				0: // Start-up/Init
					IF fbPlanarXtsMover.P_MoverSort.TrackID = GVL_General.PlanarTrackOuterFinish THEN
						fbPlanarXtsMover.P_MC_PlanarMover.MoveOnTrack(commandFeedback := fbPlanarXtsMover.P_MoverFeedback,
																			targetTrack := GVL_Mc3.MC_Tracks[E_TrackNum.Big],
																			targetPositionOnTrack := GVL_Mc3.MC_Tracks[E_TrackNum.Big].GetLength()-stTrackGlobalConfig.TargetPosnBeforeTrackEnd,
																			constraint := fbPlanarXtsMover.P_Dynamics,
																			options := fbPlanarXtsMover.P_MoverOptions.BaseMoveOptions);
						 nMoveState 	:= 20;
					ELSIF (fbPlanarXtsMover.P_MoverSort.TrackID = GVL_General.PlanarTrackOuterStart) AND 
								fbPlanarXtsMover.P_XtsPositionInfo.fPartPosition < TrackSectors.P_SectorsConfig[GC.DIVERTQ_SECTOR_OPART].PartSectorStartPosn THEN
						fbPlanarXtsMover.P_MC_PlanarMover.MoveOnTrack(commandFeedback := fbPlanarXtsMover.P_MoverFeedback,
																			targetTrack := GVL_Mc3.MC_Tracks[E_TrackNum.Main],
																			targetPositionOnTrack := GVL_Mc3.MC_Tracks[E_TrackNum.Main].GetLength()-stTrackGlobalConfig.TargetPosnBeforeTrackEnd,
																			constraint := fbPlanarXtsMover.P_Dynamics,
																			options := fbPlanarXtsMover.P_MoverOptions.BaseMoveOptions);
						 nMoveState 	:= 10;
					END_IF
					
				5: // In Recirc - from Big to Main Track - departing Gap Transition Zone - this Move command could be cyclic
					IF stPlcSystem.TempSysTime = 0 XOR stPlcSystem.TempSysTime = stPlcSystem.SysTime THEN
						stPlcSystem.TempSysTime := stPlcSystem.SysTime + (stPlcSystem.CfgIntervalExec * stPlcSystem.nCycleTime); //next valid clock to issue move command again
						fbPlanarXtsMover.P_eMerge		:= E_MergeType.NoMerge;
						fbPlanarXtsMover.P_MasterSyncId	:= 0;
						fbPlanarXtsMover.P_MasterSyncPosition	:= 0;
						fbPlanarXtsMover.P_MC_PlanarMover.MoveOnTrack(commandFeedback := fbPlanarXtsMover.P_MoverFeedback,
																		targetTrack := GVL_Mc3.MC_Tracks[E_TrackNum.Main],
																		targetPositionOnTrack := GVL_Mc3.MC_Tracks[E_TrackNum.Main].GetLength()-stTrackGlobalConfig.TargetPosnBeforeTrackEnd,
																		constraint := fbPlanarXtsMover.P_Dynamics, 
																		options := fbPlanarXtsMover.P_MoverOptions.BaseMoveOptions);
					END_IF
																		
					//Continuously call the above move command while GapInTransition TRUE (otherwise it's a one-shot command)
					IF NOT fbPlanarXtsMover.P_MoverOptions.GapInTransition THEN
						stPlcSystem.TempSysTime		:= 0;
						nMoveState 	:= 10;
					END_IF

				10: //Trig state for decision to divert
					IF TrackSectors.afbSector[GC.DIVERTQ_SECTOR_OPART].stSectorStatus.MoverEnteredSector.Q THEN
						GVL_General.stSwitchStatus.ShuttleCountAtDivertTrig		:= GVL_General.stSwitchStatus.ShuttleCountAtDivertTrig +1; //always MODing this; don't need to decrement
						TempItvlMoverIndex	:= ((GVL_General.stSwitchStatus.ShuttleCountAtDivertTrig MOD GVL_General.stSwitchConfig.SwitchModeInternal.IntervalToDivert) +1); // capture the index
					//	AllTrackSectors.M_UpdateSectorCounts(SectorNr := GC.SHORTCUT_CALC_SECTOR_IPART);
						MoverIndexDivertTrig			:= fbPlanarXtsMover.P_MoverId; // regardless of the command to divert, log the MoverID
						DivertQueue.M_UpdateAtTrig();
						nMoveState 	:= 12;
					END_IF
					
				12: // Command to move needs to be given early
					IF TrackSectors.afbSector[GC.DIVERT_DECISION_OPART].stSectorStatus.MoverEnteredSector.Q THEN
						DivertQueue.RemoveObjFromBuffer();
						nMoveState 	:= 13;
					END_IF
				
				13:				
				IF (DivertQueue.P_LastObjectRemoved.MoverID <> 0) THEN // Valid MoverID must be obtained by Remove op in previous step
					IF SwitchMagnet.P_PermIntlkOK AND NOT MagnetControlledByOtherMover AND fbPlanarXtsMover.P_CmdDivert AND 
						(fbPlanarXtsMover.P_XtsPositionInfo.fPartPosition < GVL_Mc3.TrackSectors.P_SectorConfig[GC.MAG_ON_SECTOR_OPART].PartSectorStartPosn)
						AND (stDivertingMover.SysTime <> DivertQueue.P_LastObjectRemoved.SysTime) THEN
							// Divert Move command
							stDivertingMover	:= DivertQueue.P_LastObjectRemoved;
							fbPlanarXtsMover[stDivertingMover.MoverID].P_MC_PlanarMover.MoveOnTrack(commandFeedback := fbPlanarXtsMover[stDivertingMover.MoverID].P_MoverFeedback,
																				targetTrack := GVL_Mc3.MC_Tracks[E_TrackNum.Small],
																				targetPositionOnTrack := (GVL_Mc3.MC_Tracks[E_TrackNum.Small].GetLength() - GC.SHUTTLE_LENGTH) / 2, // midpoint of shortcut
																				constraint := fbPlanarXtsMover[stDivertingMover.MoverID].P_Dynamics,
																				options := fbPlanarXtsMover[stDivertingMover.MoverID].P_MoverOptions.BaseMoveOptions);									
							nMoveState 	:= 30; //Diverting Mover
					ELSIF NOT fbPlanarXtsMover.P_CmdDivert THEN
							nMoveState 	:= 15;
					END_IF
				END_IF
	
				15: // In Recirc - from Main to Big Track
					fbPlanarXtsMover.P_MC_PlanarMover.MoveOnTrack(commandFeedback := fbPlanarXtsMover.P_MoverFeedback,
																		targetTrack := GVL_Mc3.MC_Tracks[E_TrackNum.Big],
																		targetPositionOnTrack := GVL_Mc3.MC_Tracks[E_TrackNum.Big].GetLength()-stTrackGlobalConfig.TargetPosnBeforeTrackEnd,
																		constraint := fbPlanarXtsMover.P_Dynamics,
																		options := fbPlanarXtsMover.P_MoverOptions.BaseMoveOptions);
					 nMoveState 	:= 20;				
					
				20:
					IF TrackSectors.afbSector[GC.OUTER_BIGTRACK_END].stSectorStatus.MoverEnteredSector.Q THEN
						nMoveState     := 5;
					END_IF				

				30: // Match the move command with the shuttle that is commanded to divert
					SwitchMagnet.M_EvaluateInlineCommands();
					
					IF ftMagnetControlledByOtherMover.Q THEN
						nMoveState 	:= 40;
					END_IF
			
				40: // Route through shortcut
					IF TrackSectors.afbSector[GC.LOAD_STOP_SECTOR_IPART].stSectorStatus.MoverEnteredSector.Q THEN
						IF stTrackShortcutConfig.StopAtPowerMat THEN
							nMoveState := 90;
						ELSE
							nMoveState := 50;
						END_IF					
					END_IF
					
				50: //Pre-Merge state
				IF NOT AllTrackSectors.P_AMoverIsOnSector[GC.OUTER_BIGTRACK_LSMALL] 
						(*AND stSwitchConfig.SwitchModeInternal.MaxAllowedDivertCount = GVL_General.nNumMovers*) THEN
					fbPlanarXtsMover.P_eMerge := E_MergeType.FlyingMergeMoveOnTrack;

					fbPlanarXtsMover.P_MC_PlanarMover.MoveOnTrack(commandFeedback := fbPlanarXtsMover.P_MoverFeedback,
																		targetTrack := GVL_Mc3.MC_Tracks[E_TrackNum.Small],
																		targetPositionOnTrack := GVL_Mc3.MC_Tracks[E_TrackNum.Small].GetLength()-stTrackGlobalConfig.TargetPosnBeforeTrackEnd,
																		constraint := fbPlanarXtsMover.P_Dynamics,
																		options := fbPlanarXtsMover.P_MoverOptions.BaseMoveOptions);

					nMoveState := 75;
					//Sync to Master ExpMover
				ELSIF TrackSectors.afbSector[GC.SHORTCUT_MERGE_COMMAND_FLYING].stSectorStatus.MoverEnteredSector.Q THEN
					//Nonzero means there is valid Master Mover data
					IF MergeQueue.P_LastObjectRemoved.MoverID <> 0 THEN
					fbPlanarXtsMover.P_eMerge				:= E_MergeType.FlyingMergeMoveSyncd;
						fbPlanarXtsMover.P_MasterSyncId := MergeQueue.P_LastObjectRemoved.MoverID;
//						IF MergeQueue.P_LastObjectRemoved.ExpMoverType = E_ExpMover.Head THEN
//							fbPlanarXtsMover.P_MasterSyncPosition	:= HeadExpMover[fbPlanarXtsMover.P_MasterSyncId].stExpMoverStatus.TrackSectorCenterHead;
//						ELSIF MergeQueue.P_LastObjectRemoved.ExpMoverType = E_ExpMover.Tail THEN
//							fbPlanarXtsMover.P_MasterSyncPosition	:= TailExpMover[fbPlanarXtsMover.P_MasterSyncId].stExpMoverStatus.TrackSectorCenterTail;
//						END_IF
							// use raw mover reference; likely need some position compensation, i.e, stTrackGlobalConfig.ExpMoverLength;
							fbPlanarXtsMover.P_MasterSyncPosition	:= fbPlanarXtsMover[fbPlanarXtsMover.P_MasterSyncId].P_XtsPositionInfo.fTrackPosition;							
						MergeQueue.ClearLastRemoved(); // master sync data consumed by slave
						nMoveState := 72;					
					END_IF
					
				ELSIF TrackSectors.afbSector[GC.SHORTCUT_MERGE_COMMAND_WAIT].stSectorStatus.MoverEnteredSector.Q OR 
					stTrackShortcutConfig.StopAtPowerMat THEN
					fbPlanarXtsMover.P_eMerge := E_MergeType.MergeFromStaticSyncd;
					
					fbPlanarXtsMover.P_MC_PlanarMover.MoveOnTrack(commandFeedback := fbPlanarXtsMover.P_MoverFeedback,
																		targetTrack := GVL_Mc3.MC_Tracks[E_TrackNum.Small],
																		targetPositionOnTrack := GVL_Mc3.MC_Tracks[E_TrackNum.Small].GetLength()-stTrackGlobalConfig.MergeWaitFinishDistance-stTrackGlobalConfig.MergeWaitAccelDistance,
																		constraint := fbPlanarXtsMover.P_Dynamics,
																		options := fbPlanarXtsMover.P_MoverOptions.BaseMoveOptions);

					nMoveState := 73;
				END_IF

				60: // Merge - Gear In
 //merge with gap zero
					//issue commmand to sync 
//					masterSyncPos := GVL_Mc.MC_Tracks[E_TrackNum.Big].GetLength()-100;
//					masterPosAtSync := Mover[moverInFront].MoverPos; 
//					followSyncPos := GVL_Mc.MC_Tracks[E_TrackNum.Small].GetLength()-1000;
//					followerPosAtSync :=Mover[1].MoverPos; 
//					fbMover[nForCounter].SyncToOtherMover( 
//						masterSyncPos := masterSyncPos,
//						masterTrack := GVL_Mc.MC_Tracks[E_TrackNum.Big],
//						followerSyncPos := followSyncPos,
//						followerTrack := GVL_Mc.MC_Tracks[e_TrackNum.Small],
//						PlanarMoverToFollow := fbMover[moverInFront].P_PlanarMover,
//						velo:= velo);
//						nMoveState := 80; 
//					aggressiveDynamics.SetValuesVADJ(4000,4000,8000,400000); 
//					fbMover[nForCounter].P_Dynamics := aggressiveDynamics;
					//fbMover[nForCounter].MoveOnTrack(GVL_Mc.MC_Tracks[E_TrackNum.Main],  GVL_Mc.MC_Tracks[E_TrackNum.Main].GetLength()-500,900,velo);				
				
//					IF fbPlanarXtsMover.P_eMerge <> E_MergeType.NoMerge THEN
						fbPlanarXtsMover.P_Dynamics.SetValuesVADJ(V := stMoverConfig.NormalVelo, A := stMoverConfig.MaxAccel, D := stMoverConfig.MaxDecel, J := stMoverConfig.MergeJerk);
						
						fbPlanarXtsMover.P_MC_PlanarMover.GearInPosOnTrackWithMasterMover(
								commandFeedback:= fbPlanarXtsMover.P_PlanarFeedbackGearMM, 
								masterMover:= fbPlanarXtsMover[fbPlanarXtsMover.P_MasterSyncId].P_MC_PlanarMover,
								trackTrail:= fbPlanarXtsMover.P_SyncTrail,
								masterSyncPosition:= fbPlanarXtsMover.P_MasterSyncPosition,
								masterSyncPositionTrack:= GVL_Mc3.MC_Tracks[E_TrackNum.Big], 
								slaveSyncPosition:= fbPlanarXtsMover.P_XtsPositionInfo.fTrackPosition,
								slaveSyncPositionTrack:= GVL_Mc3.MC_Tracks[E_TrackNum.Small], 
								constraint:= fbPlanarXtsMover.P_Dynamics, 
								options:= fbPlanarXtsMover.P_MoverOptions.GearInMasterMoverOptions);
								nMoveState := 74;
//					END_IF
						//fbPlanarXtsMover.P_InSync THEN				

				61:
				IF fbPlanarXtsMover.P_MoverFeedback.Done AND ManMergeCmd THEN
					ManMergeCmd	:= FALSE;
					nMoveState := 75; // 62
				END_IF
					
				62:// Permissive to Merge
//					IF NOT AllTrackSectors.P_AMoverIsOnSector[GC.OUTER_MERGE_COLLISION] THEN
//						nMoveState := 63;
//					END_IF

				63://Merge from Inner to Outer
//						fbPlanarXtsMover.P_MC_PlanarMover.MoveOnTrack(commandFeedback := fbPlanarXtsMover.P_MoverFeedback,
//																			targetTrack := GVL_Mc3.MC_Tracks[E_TrackNum.Small],
//																			targetPositionOnTrack := GVL_Mc3.MC_Tracks[E_TrackNum.Small].GetLength()-stTrackGlobalConfig.TargetPosnBeforeTrackEnd,
//																			constraint := fbPlanarXtsMover.P_Dynamics,
//																			options := fbPlanarXtsMover.P_MoverOptions.BaseMoveOptions);
//						nMoveState := 75;
				
				75: //Reset Command On Exit
						IF TrackSectors.afbSector[GC.INNER_MERGE_TO_FINISH].stSectorStatus.MoverEnteredSector.Q THEN
							stSwitchStatus.ShuttleQueueCount := stSwitchStatus.ShuttleQueueCount -1;
							nMoveState := 5;
						END_IF
				
				90: // Stopped at Powermat Station
					IF fbPlanarXtsMover.P_MoverFeedback.Done THEN
						StartTimer[nForCounter] := TRUE;
						nMoveState := 100;
					END_IF
					
				100:
					IF StopTimer[nForCounter].Q THEN
						StartTimer[nForCounter] := FALSE;
						nMoveState := 50;
					END_IF
				END_CASE
				*)

METHOD M_EvaluateTrackTransition
VAR_INPUT
	DepartingTrackRef : OTCID;
	ArrivingTrackRef : OTCID;
	DepartPermissiveSectorRef	: UDINT;
END_VAR
END_METHOD

END_FUNCTION_BLOCK

// ---- POUs/FBs/FB_RobMover.TcPOU
{attribute 'no_assign'}
FUNCTION_BLOCK FB_RobMover IMPLEMENTS I_Mover
VAR_INPUT
END_VAR
VAR_OUTPUT
END_VAR
VAR
	fbPlanarMover : MC_PlanarMover;
	fbPlanarFeedback: MC_PlanarFeedback;
	CmdFeedback :  XtsCommandFeedback;
	bIsInitialized: BOOL;
	ipXtsMover:   I_XtsXlMover1;
	ipXtsProcessingUnit:  I_XtsProcessingUnit1;
	trackTrail: MC_PlanarTrackTrail;
	nextMcTrackOid: OTCID;
	stMoveOnTrackOptions: ST_MoveOnTrackOptions;
	_stDynamics: DynamicConstraint_PathXY;
	_TargetTrack : UDINT;
	_ReWork : BOOL;
	partConfig1: UINT;
	SyncMoverFeedback: Tc3_Mc3PlanarMotion.MC_PlanarFeedbackGearInPosOnTrackWithMasterMover;
	_InSync :BOOL; 
	options: Tc3_Mc3PlanarMotion.ST_GearInPosOnTrackWithMasterMoverOptions;
	syncTrail : MC_PlanarTrackTrail; 
END_VAR

METHOD CycleUpdate : BOOL
VAR_INPUT
END_VAR
IF NOT bIsInitialized THEN
	RETURN;
END_IF

fbPlanarMover.GetTrackTrailInformation(trackTrail);


fbPlanarMover.Update();


fbPlanarFeedback.Update();
SyncMoverFeedback.Update(); 
_InSync := SyncMoverFeedback.inSync; 

UpdateXtsTrack();
END_METHOD

METHOD Init : BOOL
VAR_INPUT

	XtsMover:   I_XtsXlMover1;
	XtsProcessingUnit :  I_XtsProcessingUnit1;
END_VAR



ipXtsMover:= XtsMover;
ipXtsProcessingUnit :=  XtsProcessingUnit;

stMoveOnTrackOptions.direction := MC_Direction.mcDirectionPositive;
stMoveOnTrackOptions.gapMode := MC_GAP_MODE_ON_TRACK.Fast1D;
stMoveOnTrackOptions.gap:= 800;

syncTrail.AddTrack(track:= GVL_Mc.MC_Tracks[E_TrackNum.Small]); 
syncTrail.AddTrack(track:= GVL_Mc.MC_Tracks[E_TrackNum.Main]); 


//_stDynamics.SetValuesVADJ(500, 4000, 4000, 10000);

bIsInitialized := TRUE;
END_METHOD

METHOD JoinNearestTrack : BOOL


VAR_INST
	nForCounter: UINT;
	mcTrackOid: OTCID;
	partOid: OTCID;
	cmdFeedback					: 	XtsCommandFeedback;
	objectInfo: PlanarObjectInfo;
END_VAR
partOid := ipXtsMover.GetPositionInfo_partObjectId(cmdFeedback);

IF partOid = 0 THEN
	RETURN;
END_IF

IF cmdFeedback.IsDone THEN
	mcTrackOid := ipXtsProcessingUnit.XlPartWithOid(partOid, cmdFeedback).GetMcTrackOid(cmdFeedback);
	
	FOR nForCounter := 1 TO GVL_MC.nTrackCount DO
		objectInfo := GVL_MC.Mc_Tracks[nForCounter].GetPlanarObjectInfo();
		IF objectInfo.Id = mcTrackOid THEN
			fbPlanarMover.JoinTrack(fbPlanarFeedback, GVL_MC.Mc_Tracks[nForCounter], _stDynamics, 0); 
			RETURN;
		END_IF
	END_FOR
END_IF
END_METHOD

METHOD LeaveSystemAt : BOOL
VAR_INPUT
	ConnectionOut: REFERENCE TO MC_PlanarTrackConnectionOut;
END_VAR
fbPlanarMover.LeaveSystemAt(fbPlanarFeedback, ConnectionOut,  _stDynamics,0);
END_METHOD

METHOD MoveOnTrack : BOOL
VAR_INPUT
	
	track: REFERENCE TO MC_PlanarTrack;	
	targetPos: LREAL;
	gap : LREAL; 
	velo : LREAL; 
END_VAR
stMoveonTrackOptions.gap := gap; 
THIS^.P_Dynamics.V := velo; 
fbPlanarMover.MoveOnTrack(fbPlanarFeedback, track, targetPos, _stDynamics, stMoveOnTrackOptions);
END_METHOD

PROPERTY MoverOTCID : OTCID
GET
MoverOTCID := fbPlanarMover.MCTOPLC.STD.MoverOID;
END_GET
SET
END_SET
END_PROPERTY

PROPERTY MoverStopped : BOOL
GET
MoverStopped := (fbPlanarMover.MCTOPLC.SETONTRACK.SetVelo < 20);
END_GET
SET
END_SET
END_PROPERTY

PROPERTY P_Dynamics : REFERENCE TO DynamicConstraint_PathXY;
GET

P_Dynamics REF= _stDynamics;
END_GET
SET // PUBLIC
_stDynamics := P_Dynamics;
END_SET
END_PROPERTY

PROPERTY P_InSync : Bool
GET
P_InSync := _InSync;
END_GET
END_PROPERTY

PROPERTY P_PlanarFeedback : REFERENCE TO MC_PlanarFeedback
GET
P_PlanarFeedback REF= fbPlanarFeedback;
END_GET
END_PROPERTY

PROPERTY P_PlanarMover :   REFERENCE TO  MC_PlanarMover
GET
P_PlanarMover REF= fbPlanarMover;
END_GET
END_PROPERTY

PROPERTY P_TargetTrack : UDINT
GET
P_TargetTrack := _TargetTrack ;
END_GET
SET
_TargetTrack := P_TargetTrack;
END_SET
END_PROPERTY

PROPERTY Rework : BOOL
GET
Rework := _Rework;
END_GET
SET
_Rework := Rework;
END_SET
END_PROPERTY

METHOD SyncToOtherMover : BOOL
VAR_INPUT
	masterSyncPos : LREAL; // Position on the master track
	followerSyncPos : LREAL; // position on the follower track
	PlanarMoverToFollow: REFERENCE TO Tc3_Mc3PlanarMotion.MC_PlanarMover;
	masterTrack : REFERENCE TO Tc3_Mc3PlanarMotion.MC_PlanarTrack; 
	followerTrack : REFERENCE TO Tc3_Mc3PlanarMotion.MC_PlanarTrack; 
	velo : LREAL; 
END_VAR

VAR
	trail: Tc3_Mc3PlanarMotion.MC_PlanarTrackTrail;

END_VAR
Options.allowedSlaveSyncDirections := MC_SYNC_DIRECTIONS.Positive; 
options.directionMasterSyncPosition := MC_DIRECTION.mcDirectionNonModulo; 
options.directionSlaveSyncPosition := MC_DIRECTION.mcDirectionNonModulo;  
options.followMover := FALSE; 
options.gap := 0; // elimnate gap funciton 
options.inSyncToleranceDistance :=0; 
options.moduloToleranceMasterSyncPosition := 0; 
options.moduloToleranceSlaveSyncPosition := 0;  
_stDynamics.V := velo; 

fbPlanarMover.GearInPosOnTrackWithMasterMover(
	commandFeedback:=  SyncMoverFeedback , 
	masterMover:= PlanarMoverToFollow , 
	trackTrail:= syncTrail, // may need to give a trail maybe not
	masterSyncPosition:= masterSyncPos, 
	masterSyncPositionTrack:= MasterTrack , 
	slaveSyncPosition:= followerSyncPos, 
	slaveSyncPositionTrack:= followerTrack, 
	constraint:=_stDynamics , 
	options:=options );
END_METHOD

METHOD PUBLIC UpdateXtsTrack
VAR_INPUT
END_VAR
VAR_STAT
	nTrackCount: UINT;
	oid1: OTCID;
	oid2: OTCID;
	
	nForCounter: UINT;
	nPartConfigCount: UINT;
	
	partConfig1: OTCID;
	partConfig2: OTCID;
	
	mcTrackOid1: OTCID;
	mcTrackOid2: OTCID;
	trackOid: OTCID;
	
	nTrackTrailCount: UDINT;
	actTrackOid: OTCID;
	nIndexInTrail: UDINT;
END_VAR
nTrackTrailCount := trackTrail.TrackCount;
actTrackOid := fbPlanarMover.MCTOPLC.SETONTRACK.TrackOID;

IF nTrackTrailCount <= 1 THEN
	RETURN;
END_IF

FOR nForCounter := 1 TO UDINT_TO_UINT(nTrackTrailCount) DO
	oid1 := trackTrail.GetTrackOidAt(nForCounter);
	IF oid1 = actTrackOid THEN
		IF nForCounter < nTrackTrailCount THEN
			oid2 := trackTrail.GetTrackOidAt(nForCounter + 1);
			EXIT;
		ELSE
			RETURN; //last one ine track trail
		END_IF
	END_IF
END_FOR

IF oid2 = nextMcTrackOid AND   ipXtsMover.GetPositionInfo_partPosition(CmdFeedback) < 600THEN //no change
	RETURN;
END_IF

nTrackCount := ipXtsProcessingUnit.TrackCount();

FOR nForCounter := 1 TO nTrackCount DO
	nPartConfigCount := ipXtsProcessingUnit.Track(nForCounter, CmdFeedback).PartConfigCount(); 
	
	IF nPartConfigCount >= 2  THEN
		partConfig1 := ipXtsProcessingUnit.Track(nForCounter, CmdFeedback).GetPartConfigOidAt(1, 0);
		partConfig2 := ipXtsProcessingUnit.Track(nForCounter, CmdFeedback).GetPartConfigOidAt(2, 0);
//
		
		IF partConfig1 = 0 OR partConfig2 = 0 THEN
			CONTINUE;
		END_IF
		
		mcTrackOid1 := ipXtsProcessingUnit.XlPartWithOid(partConfig1, CmdFeedback).GetMcTrackOid(0);
		mcTrackOid2 := ipXtsProcessingUnit.XlPartWithOid(partConfig2, CmdFeedback).GetMcTrackOid(0);
		IF mcTrackOid1 = oid1 AND mcTrackOid2 = oid2   THEN
			trackOid := ipXtsProcessingUnit.Track(nForCounter, CmdFeedback).GetObjectId();
			ipXtsMover.SetActiveTrackObjectId(trackOid, CmdFeedback);
			
			IF CmdFeedback.IsDone THEN
				nextMcTrackOid := oid2;
			END_IF
			
			RETURN;
		END_IF
	END_IF
END_FOR
END_METHOD

PROPERTY XlProcessingUnit : I_XtsProcessingUnit1
GET
XlProcessingUnit := ipXtsProcessingUnit;
END_GET
END_PROPERTY

PROPERTY XtsComFeed : REFERENCE TO  XtsCommandFeedback
GET
XtsComFeed REF= CmdFeedback;
END_GET
END_PROPERTY

PROPERTY XtsXlMover : I_XtsXlMover1
GET
XtsXlMover := ipXtsMover;
END_GET
END_PROPERTY

END_FUNCTION_BLOCK

// ---- POUs/FBs/ReadTcCom.TcPOU
FUNCTION_BLOCK ReadTcCom
VAR_INPUT
	
END_VAR
VAR_OUTPUT
	bBusy 				: BOOL;
	bDone 				: BOOL;
	bError 				: BOOL;
	bGetComObject	: BOOL;
END_VAR
VAR
	
	_nObjectId				: OTCID;
	_ipComObject 			: ITComObject;
	_nSoftDriveOid			: OTCID;
	PID_Value	: PTCID := 	16#05030149;
END_VAR

METHOD GetComObject : BOOL
VAR_INPUT
	nObjectId	: OTCID;
END_VAR
IF FW_ObjMgr_GetObjectInstance(	oid		:= nObjectId, 
								iid		:= TC_GLOBAL_IID_LIST.IID_ITComObject, 
								pipUnk	:= ADR(_ipComObject)) = 0
THEN
	GetComObject := TRUE;
END_IF
END_METHOD

METHOD GetValue : ARRAY[1..nNumMovers] OF OTCID
VAR_INPUT
	PID_Value 		: otcid;
END_VAR
VAR
	Value			: ARRAY[1..nNumMovers] OF OTCID;
	nData 			: UDINT := SIZEOF(Value);
	pData 			: PVOID := ADR(Value);
	stEventEntry	: TcEventEntry;
	pstEventEntry	: REFERENCE TO TcEventEntry REF= stEventEntry;
	
END_VAR
VAR_INST
	hResult : HRESULT;
END_VAR
IF _ipComObject <> 0  THEN
	 hResult := _ipComObject.TcGetObjPara(
				pid 	:= PID_Value,
				nData 	:= nData,
				pData 	:= pData,
				pgp   	:=0) ;
	IF hResult = 0	THEN
		GetValue := Value;
		bError := FALSE;
	ELSE
		bError := TRUE;
	END_IF
END_IF
END_METHOD

END_FUNCTION_BLOCK

// ---- POUs/FUNs/F_t_v0.TcPOU
FUNCTION F_t_v0 : TIME
VAR_INPUT
	PosnDelta	: LREAL;
	Accel		: LREAL;
END_VAR
VAR
END_VAR

IF Accel <> 0 THEN
	F_t_v0	:= LREAL_TO_TIME(SQRT((2*PosnDelta)/Accel));
END_IF

END_FUNCTION

// ---- POUs/FUNs/F_t_vConstant.TcPOU
FUNCTION F_t_vConstant : TIME
VAR_INPUT
	Velo		: LREAL;
	PosnDelta	: LREAL;
END_VAR

IF Velo <> 0 THEN
	F_t_vConstant	:= LREAL_TO_TIME (PosnDelta / Velo);
END_IF

END_FUNCTION

// ---- POUs/FUNs/PositionF_CurrentCoeff.TcPOU
FUNCTION PositionF_CurrentCoeff : LREAL
VAR_INPUT
    Current : LREAL;
END_VAR
VAR
END_VAR

PositionF_CurrentCoeff   := (-0.0009*Current)+ 1.0016;

END_FUNCTION
